{attribute 'qualified_only'}
VAR_GLOBAL
//Heartbeat
	benable_heartbeat:		BOOL; //for groundstation output
	bheartbeat_OK: 			BOOL := TRUE; //for groundstation evaluation
	
	bprecharge:				BOOL;
	
	
	bsdc_closed:				BOOL;
 
	bengage_brakes AT %Q*:			BOOL := FALSE; //Normally Closed system -> TRUE when retracted False when engaged
	bCLKTrigger AT %Q*:				BOOL := FALSE; 
	bbrakes_engaged AT %I*:			BOOL := FALSE; //Normally Closed system -> TRUE when retracted False when engaged
	
	bsafety_inputs_valid AT %I*: 	BOOL; //done through twinsafe PLC-TWINSAFE Run mode verification
	
	b_EmergencyLine AT %Q*: 			BOOL := TRUE; //NC System

	bEstopError:				BOOL; 
	bEstopRestart:			BOOL := FALSE; //Used to restart the Estop from the PLC 
	bEstopRestartTracker:	BOOL := FALSE;
	
	benable_telemetry: 		BOOL;
	
	bcan_bus_ok: 			BOOL := TRUE; 
	nMasterDevStateCouplers AT %I*: UINT; 
	nMasterDevStatePLC AT %I*: UINT; 
	bethercat_ready:  		BOOL; 
	
	
	
	//Critical Temperatures for Shutdown
	rcritical_temp_prop: 	REAL := 100.0; //maximum allowable temperature for propulsion. STILL A GUESS!!!!!
	rcritical_temp_HEMS: 	REAL := 40.0; //maximum allowable temperature for levitation HEMS
	rcritical_temp_EMS:		REAL := 60.0; //maximum allowable temperature for levitation EMS
	rcritical_temp_watercooling:	REAL;
	//rcritical_temp_PT:		REAL; //maximum allowable temperature for powertrain. commented out for now because PT should do this themselves
	
	
	//Temperatures to re enable after cooldown
	rcritical_temp_prop_coolDown: 	REAL := 95.0; //maximum allowable temperature for propulsion. STILL A GUESS!!!!!
	rcritical_temp_HEMS_coolDown: 	REAL := 35.0; //maximum allowable temperature for levitation HEMS
	rcritical_temp_EMS_coolDown:		REAL := 55.0; //maximum allowable temperature for levitation EMS
	rcritical_temp_watercooling_coolDown:	REAL;
	rcritical_temp_PT_coolDown:		REAL; //maximum allowable temperature for powertrain. commented out for now because PT should do this themselves
	

END_VAR

(* stored: Version 1.1.0.1
   GVL GVL_FSM: Id {e9f32245-b0fa-4870-9fb8-012882e1d02d} *)
